(* CODESYS project Ethercat_read_write_parameter_V1.1.export

Project tree, tasks and I/O mapping:
  function block read_ETC_DRV28 [LD]
  function block write_ETC_DRV [LD]
*)

// read_ETC_DRV28
FUNCTION_BLOCK read_ETC_DRV28
VAR_INPUT
	stop: BOOL;
	slave_ID: UINT;
	Group_param: WORD;
	Sub_Group_param: BYTE;
	
END_VAR
VAR_OUTPUT
	busy: BOOL;
	error: BOOL;
	er_code: ETC_CO_ERROR;
	value_param: WORD;
END_VAR
VAR
	Sub_Index: BYTE;
	wIndex: WORD;
	read: BOOL;
	TON_1: TON;
	sdo_Read_1: ETC_CO_SdoRead4;
	abort: UDINT;
	read_data: ARRAY [1..4] OF BYTE;
	lenght: USINT;
	done: BOOL;
END_VAR
VAR // added by the converter: edge detectors and wires of the graphical bodies
    _w1 : BOOL;
END_VAR

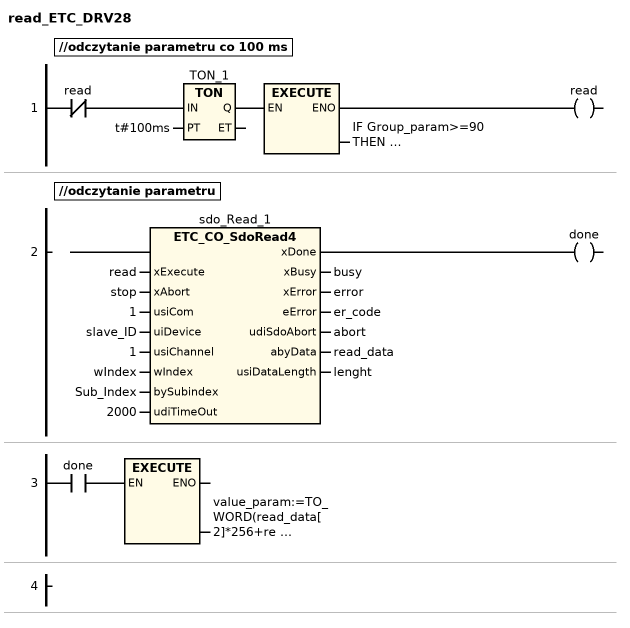
// NETWORK 1
// label: //odczytanie parametru co 100 ms
TON_1(IN := NOT read, PT := t#100ms); // TON
_w1 := TON_1.Q;
IF _w1 THEN
    IF Group_param>=90 THEN
    	wIndex:=Group_param+16#1FC3;
    ELSE
    	wIndex:=Group_param+16#2000;
    END_IF
    
    Sub_Index:=Sub_Group_param+1;
END_IF
read := _w1;

// NETWORK 2
// label: //odczytanie parametru
sdo_Read_1(
    xExecute := read,
    xAbort := stop,
    usiCom := 1,
    uiDevice := slave_ID,
    usiChannel := 1,
    wIndex := wIndex,
    bySubindex := Sub_Index,
    udiTimeOut := 2000,
    xBusy => busy,
    xError => error,
    eError => er_code,
    udiSdoAbort => abort,
    abyData => read_data,
    usiDataLength => lenght); // ETC_CO_SdoRead4
done := sdo_Read_1.xDone;

// NETWORK 3
IF done THEN value_param:=TO_WORD(read_data[2]*256+read_data[1]); END_IF

// NETWORK 4

END_FUNCTION_BLOCK

// write_ETC_DRV
FUNCTION_BLOCK write_ETC_DRV
VAR_INPUT
	Value: INT;
	stop: BOOL;
	slave_ID: UINT;
	Group_param: WORD;
	Sub_Group_param: BYTE;
END_VAR
VAR_OUTPUT
	busy: BOOL;
	error: BOOL;
	er_code: ETC_CO_ERROR;
END_VAR
VAR
	wIndex: WORD;
	Sub_Index: BYTE;
	data_array: ARRAY [1..4] OF BYTE;
	save: BOOL;
	SDO_write: ETC_CO_SdoWrite4;
	abort: UDINT;
END_VAR

VAR_IN_OUT
	write: BOOL;
END_VAR
VAR // added by the converter: edge detectors and wires of the graphical bodies
    _w1 : BOOL;
END_VAR

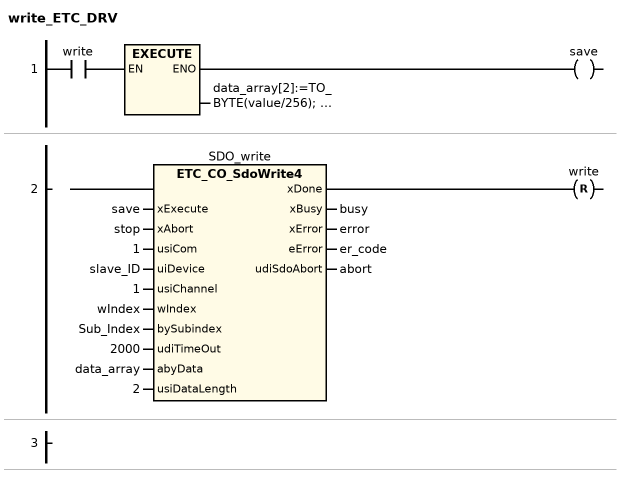
// NETWORK 1
_w1 := write;
IF _w1 THEN
    data_array[2]:=TO_BYTE(value/256);
    data_array[1]:=TO_BYTE(Value-TO_INT(data_array[2]*256));
    IF Group_param>=90 THEN
    	wIndex:=Group_param+16#1FC3;
    ELSE
    	wIndex:=Group_param+16#2000;
    END_IF
    	Sub_Index:=Sub_Group_param+1;
END_IF
save := _w1;

// NETWORK 2
SDO_write(
    xExecute := save,
    xAbort := stop,
    usiCom := 1,
    uiDevice := slave_ID,
    usiChannel := 1,
    wIndex := wIndex,
    bySubindex := Sub_Index,
    udiTimeOut := 2000,
    abyData := data_array,
    usiDataLength := 2,
    xBusy => busy,
    xError => error,
    eError => er_code,
    udiSdoAbort => abort); // ETC_CO_SdoWrite4
write R= SDO_write.xDone;

// NETWORK 3

END_FUNCTION_BLOCK
